PROGRAM Main
VAR
	promise_TestSuite : Promise_TestSuite;
END_VAR

TcUnit.Run();

END_PROGRAM

(* stored: Version 1.1.0.1, ProductVersion 3.1.4026.6
   POU Main: Id {55dc8056-a83c-498b-9d09-689d30efbd92}, SpecialFunc None *)
